FUNCTION_BLOCK FB_ToggleSwitch
VAR_INPUT
	switch : BOOL;
END_VAR
VAR_OUTPUT
	status : BOOL;
END_VAR
VAR
	pEdge : BOOL;
END_VAR


IF switch AND NOT pEdge THEN
	pEdge := TRUE;
	IF NOT status THEN
		status := TRUE;
	ELSE
		status := FALSE;
	END_IF
END_IF

pEdge := switch;

END_FUNCTION_BLOCK

(* stored: Version 1.1.0.1, ProductVersion 3.1.4022.18
   POU FB_ToggleSwitch: Id {bd8adc6a-b93b-471d-8430-b3f1af2cbb49}, SpecialFunc None *)
